// SIMATIC S7-200 project (STEP 7-Micro/WIN), CPU 224 REL 02.01

ORGANIZATION_BLOCK MAIN:OB1
TITLE=PROGRAM COMMENTS
BEGIN
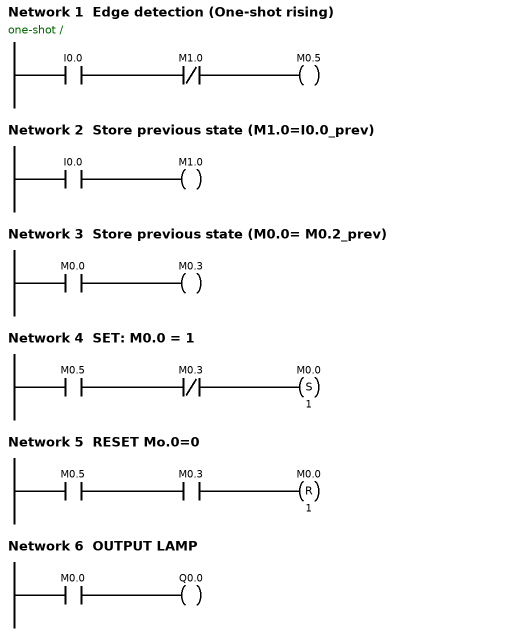
Network 1 // Edge detection (One-shot rising)
// one-shot
// 
LD     I0.0
AN     M1.0
=      M0.5
Network 2 // Store previous state (M1.0=I0.0_prev)
LD     I0.0
=      M1.0
Network 3 // Store previous state (M0.0= M0.2_prev)
LD     M0.0
=      M0.3
Network 4 // SET: M0.0 = 1
LD     M0.5
AN     M0.3
S      M0.0, 1
Network 5 // RESET Mo.0=0
LD     M0.5
A      M0.3
R      M0.0, 1
Network 6 // OUTPUT LAMP
LD     M0.0
=      Q0.0
END_ORGANIZATION_BLOCK
